FUNCTION proj9_TupleStruct_1: REAL
{ S7_Optimized_Access := 'false' }
    VAR_INPUT
        tuple: TupleStruct_1;
    END_VAR

BEGIN
    proj9_TupleStruct_1 := tuple.field9;
END_FUNCTION
